// TIA Portal V21 export
DATA_BLOCK "AUXILIARY"   // DB6
{ S7_Optimized_Access := 'TRUE' }
// stored: MemoryReserve 100
   VAR
      PULSE : Array[0..40] of Bool;
      "PWD STEAM ON" : Bool := TRUE;
      "CHAMBER TEMP" : Real := 0.0;
      "CHAMBER PRESS" : Real := 0.0;
      "START VACCUM" : Real := 0.0;
      "END VACCUM" : Real := 0.0;
      "ACTUAL LEAK" : Real := 0.0;
   END_VAR
   VAR RETAIN
      "STD TEMP1" : Real := 114.0;
      "STD TEMP2" : Real := 116.0;
      "STD TEMP3" : Real := 119.0;
      "STD PRESS" : Real := 0.1;
      "STD HOLD1" : Int := 5;
      "STD HOLD2" : Int := 3;
      "STD HOLD3" : Int := 2;
      "STD VCC" : Real := 0.0;
      "STD UP PRESS" : Real := 0.0;
      "STD VCC HOLD" : Int := 0;
      "NO OF STD PULSE" : Int := 0;
   END_VAR
   VAR
      "DRUM VFD" : Real := 8192.0;
      "STR STEAM ON" : Bool := FALSE;
      PULSE1 : Array[0..50] of Bool;
      pulse2 : Array[0..50] of Bool;
   END_VAR
   VAR RETAIN
      "STERILE HOLD TEMP" : Real := 121.4;
      "STERILE HOLD TIME" : Int := 30;
      "CONTROL BAND" : Real := 0.0;
      "STERILE STOP TEMP" : Real := 120.9;
   END_VAR
   VAR
      "STD CRITICAL TEMP" : Real;
   END_VAR
BEGIN
   PULSE[0..40] := FALSE;
   PULSE1[0..50] := FALSE;
   pulse2[0..50] := FALSE;
END_DATA_BLOCK
